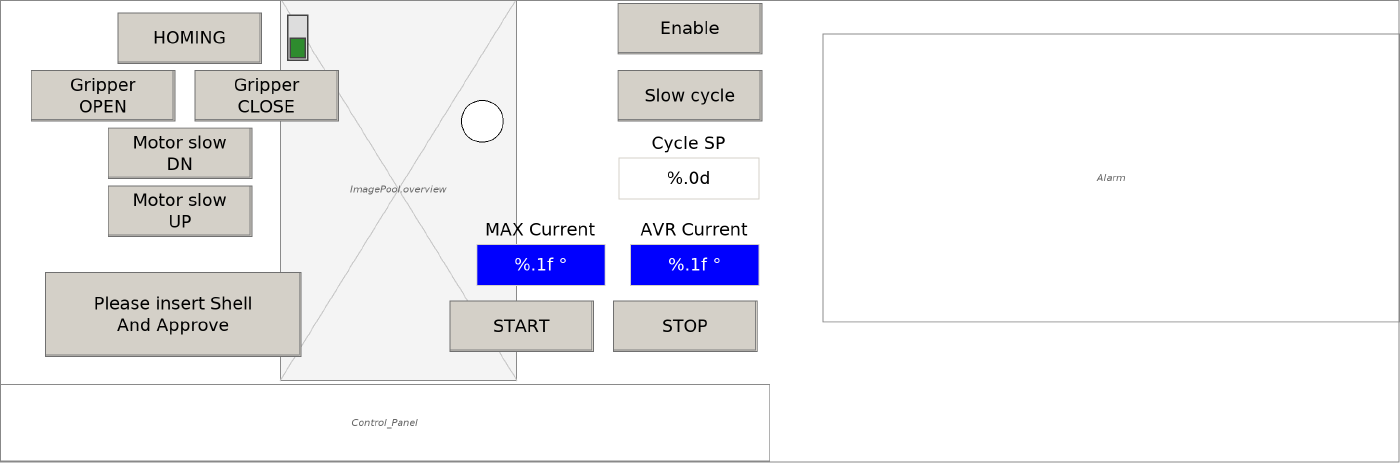
VISUALIZATION Overview_ATP  // 1455x482
    Button (122,13 150x53), "HOMING", colour toggle: GVL_IO.Homing_OK
        tap GVL_IO.Homing
    Button (32,73 150x53), "Gripper OPEN", colour toggle: GVL_IO.test_Gripper_open_OK, invisible if: not GVL_IO.Homing_OK
        tap GVL_IO.Gripper_Open_cmd
    Button (112,193 150x53), "Motor slow UP", colour toggle: GVL_IO.test_motor_slUP_ok, invisible if: not GVL_IO.Homing_OK
        tap GVL_IO.Motor_UP_slow_cmd
    Button (112,133 150x53), "Motor slow DN", colour toggle: GVL_IO.test_motor_sldown_ok, invisible if: not GVL_IO.Homing_OK
        tap GVL_IO.Motor_DN_slow_cmd
    Frame (0,400 800x80)
        shows Control_Panel()
    Image (291,-2 246x398), image: ImagePool.overview
    Label (206,13 131x32)
    Button (467,313 150x53), "START", invisible if: not GVL_IO.Homing_OK
        tap GVL_IO.ATP_start_cmd
    Button (637,313 150x53), "STOP", colour toggle: GVL_IO.Stop
        tap GVL_IO.Stop
    Ellipse (479,104 44x44), colour toggle: GVL_IO.ixHome_Position
    Button (202,73 150x53), "Gripper CLOSE", colour toggle: GVL_IO.test_Gripper_close_OK, invisible if: not GVL_IO.Homing_OK
        tap GVL_IO.Gripper_Close_cmd
    Button (642,3 150x53), "Enable", colour toggle: GVL_IO.qxSTO_toDrive
        OnMouseClick: toggle GVL_IO.Enable_motor_cmd
    Button (47,283 266x88), "Please insert Shell And Approve", colour toggle: GVL_IO.test_Insert_OK, invisible if: not GVL_IO.Homing_OK
        toggle GVL_IO.test_Insert_OK
    Button (642,73 150x53), "Slow cycle", colour toggle: GVL_IO.test_slowCycle_OK, invisible if: not GVL_IO.Homing_OK
        tap GVL_IO.Slow_cycle_cmd
    Label (644,133 143x32), "Cycle SP", invisible if: not GVL_IO.Homing_OK
    Textfield (643,164 146x43), "%.0d", text variable: GVL_IO.Cycle_SP, invisible if: not GVL_IO.Homing_OK
        OnMouseClick: write the text variable via Default
    Label (496,223 131x32), "MAX Current"
    Textfield (495,254 134x43), "%.1f °", text variable: GVL_IO.Motor_I_MAX
    Label (656,223 131x32), "AVR Current"
    Textfield (655,254 134x43), "%.1f °", text variable: GVL_IO.Motor_I_AVR
    DipSwitch (283,15 53x48), variable: GVL_IO.Homing_OK, behaviour: TOGGLE, style: Switch-DipSwitch-Green
    Frame (855,35 600x300), invisible if: GVL_IO.Error = 0
        shows Alarm()
        p3560616238: -750
END_VISUALIZATION

(* stored: Version 1.1.0.1, ProductVersion 3.1.4024.15
   Visu Overview_ATP: Id {20f0529a-4252-4240-a646-c547253f7162} *)
